# EPICS substitutions: ioc/iocBoot/iocsm/Db/backup/galil_motor_extras.substitutions
# $File: //ASP/Dev/SBS/4_Controls/4_3_Network_Infrastructure/4_3_1_Comms_Common_Services/sw/device_drivers/Galil/1-5/galilTestApp/Db/galil_motor_extras.substitutions $
# $Revision: #3 $
# $DateTime: 2012/03/22 09:46:31 $
# $Author: cliftm $
#
# Description
# Substitution file for readback/commands that are in addition to features provided by motorRecord
#
# This library is free software; you can redistribute it and/or
# modify it under the terms of the GNU Lesser General Public
# Licence as published by the Free Software Foundation; either
# version 2.1 of the Licence, or (at your option) any later version.
#
# This library is distributed in the hope that it will be useful,
# but WITHOUT ANY WARRANTY; without even the implied warranty of
# MERCHANTABILITY or FITNESS FOR A PARTICULAR PURPOSE.  See the GNU
# Lesser General Public Licence for more details.
#
# You should have received a copy of the GNU Lesser General Public
# Licence along with this library; if not, write to the Free Software
# Foundation, Inc., 51 Franklin St, Fifth Floor, Boston, MA 02110-1301 USA.
#
# Contact details:
# mark.clift@synchrotron.org.au
# 800 Blackburn Road, Clayton, Victoria 3168, Australia.
#
# P - Motion device
# M - Motor name
# PORT - Asyn port of controller
# ADDR - Axis number 0-7
# PREC - Precision of analog records
# SCAN - Scan period for monitor records.  Use passive when only epics will change value (default)
#      - Periodic scan will slow controller update performance (poller)
# MTRTYPE - motor type =
#       	0 - Servo
#		1 - Reverse servo
#		2 - High active stepper
#		3 - Low active stepper
#		4 - Reverse high active stepper
#		5 - Reverse low active stepper
# MTRON - motor off 0, motor on 1

file "$(GALIL)/GalilSup/Db/galil_motor_extras.template"
{
pattern
{   P,       M,    PORT,    ADDR, PREC, SCAN,       MTRTYPE, MTRON, EGU  }
 {  "X14B1:EX:Diff", "Phi",  "Galil2183", 0,    5,    "Passive",  "3",     "0",   "deg" }
 {  "X14B1:EX:Diff", "B",    "Galil2183", 1,    5,    "Passive",  "0",     "0",   "deg" }
 {  "X14B1:EX:Diff", "TTH",   "Galil2183", 2,    5,    "Passive",  "3",     "0",   "deg" }
 {  "X14B1:EX:Diff", "D",    "Galil2183", 3,    5,    "Passive",  "3",     "0",   "deg" }
 {  "X14B1:EX:Diff", "TH",    "Galil2183", 4,    5,    "Passive",  "3",     "0",   "deg" }
 {  "X14B1:EX:CCD", "X",    "Galil2183", 5,    5,    "Passive",  "5",     "0",   "mm" }
 {  "X14B1:EX:CCD", "Y",    "Galil2183", 6,    5,    "Passive",  "5",     "0",   "mm" }
 {  "X14B1:EX:CCD", "Z",    "Galil2183", 7,    5,    "Passive",  "5",     "0",   "mm" }
}

# end
